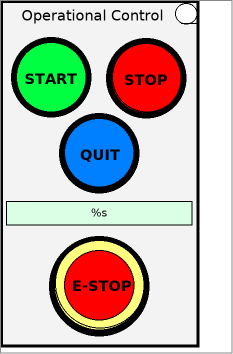
VISUALIZATION OperationalControlPad  // 233x354
VAR_IN_OUT
	stVisOperationalControl	: ST_Vis_OperationalControl;
END_VAR
    Rectangle (0,0 199x347)
    Label (9,1 167x29), "Operational Control"
    Ellipse (11,37 80x80)
    Ellipse (16,42 70x70)
    Ellipse (16,42 70x70), invisible if: NOT stVisOperationalControl.bStartButtonLamp
    Ellipse (106,38 80x80)
    Ellipse (111,43 70x70)
    Ellipse (111,43 70x70), invisible if: Not stVisOperationalControl.bStopButtonLamp
    Ellipse (59,113 80x80)
    Ellipse (64,118 70x70)
    Ellipse (64,118 70x70), invisible if: NOT stVisOperationalControl.bQuitButtonLamp
    Label (13,64 76x30), "START"
    Label (108,65 76x30), "STOP"
    Label (62,140 76x30), "QUIT"
    Rectangle (6,201 186x24), "%s", text variable: stVisOperationalControl.sMessage
    Ellipse (49,236 100x100)
    Ellipse (54,240 90x90)
    Ellipse (64,250 70x70)
    Ellipse (64,250 70x70), invisible if: NOT stVisOperationalControl.bEStopButtonLamp
    Label (64,271 76x30), "E-STOP"
    Rectangle (6,201 186x24), "%s", text variable: stVisOperationalControl.sMessage, invisible if: NOT stVisOperationalControl.bMessageColorRed
    Rectangle (6,201 186x24), "%s", text variable: stVisOperationalControl.sMessage, invisible if: NOT stVisOperationalControl.bMessageColorGreen
    Ellipse (16,42 70x70)
        tap stVisOperationalControl.bStartButtunState
    Ellipse (112,42 70x70)
        tap stVisOperationalControl.bStopButtonState
    Ellipse (64,117 70x70)
        tap stVisOperationalControl.bQuitButtonState
    Ellipse (55,238 90x90)
        toggle stVisOperationalControl.bEStopButtonState
    Ellipse (175,3 22x21)
    Line (218,-7) (233,-6)
    Line (181,23) (197,23)
    Rectangle (158,2 40x30)
        OnMouseClick: execute { stVisOperationalControl.bVisInvisibleButton := TRUE; }
END_VISUALIZATION

(* stored: Version 1.1.0.1, ProductVersion 3.1.4024.9
   Visu OperationalControlPad: Id {ab730b08-ca29-490a-9aa6-03fd929ed4ce} *)
